TYPE E_SwivelCtrl :
(
	Original,
    Swiveled
)USINT;
END_TYPE

(* stored: Version 1.1.0.1, ProductVersion 3.1.4020.6
   DUT E_SwivelCtrl: Id {300b88fb-6e9c-4e7c-89bd-02b13af7ce39} *)
